(* IEC 61131-3 sources: matiec/tests/cli/profile-fixtures, 26 files *)

(* ---- namespace-internal-local.st ---- *)
NAMESPACE INTERNAL Secret
TYPE
  Value : INT;
END_TYPE

FUNCTION Identity : Value
  VAR_INPUT
    Input : Value;
  END_VAR
  Identity := Input;
END_FUNCTION
END_NAMESPACE

(* ---- reference-local-lifetime.st ---- *)
FUNCTION REFERENCE_LOCAL_LIFETIME_TEST : INT
  VAR
    VALUE : INT;
    VALUE_REF : REF_TO INT;
  END_VAR

  VALUE := 7;
  VALUE_REF := REF(VALUE);
  REFERENCE_LOCAL_LIFETIME_TEST := VALUE_REF^;
END_FUNCTION

(* ---- object-method-nested.st ---- *)
FUNCTION_BLOCK NestedCounter
  VAR Count : INT := 0; END_VAR
  Count := Count;

  METHOD PUBLIC Increment : INT
    VAR_INPUT Delta : INT; END_VAR
    Count := Count + Delta;
    Increment := Count;
  END_METHOD
END_FUNCTION_BLOCK

PROGRAM NestedDemo
  VAR
    Instance : NestedCounter;
    Result : INT;
  END_VAR
  Result := Instance.Increment(Instance.Increment(1));
END_PROGRAM

(* ---- object-method-private.st ---- *)
FUNCTION_BLOCK Counter
  VAR
    Count : INT;
  END_VAR
  Count := Count;

  METHOD PRIVATE Hidden : INT
    Hidden := Count;
  END_METHOD
END_FUNCTION_BLOCK

(* ---- object-method-unknown.st ---- *)
FUNCTION_BLOCK Counter
  VAR
    Count : INT;
  END_VAR
  Count := Count;

  METHOD PUBLIC Increment : INT
    Increment := Count;
  END_METHOD
END_FUNCTION_BLOCK

PROGRAM BadMethod
  VAR
    CounterInstance : Counter;
    Result : INT;
  END_VAR
  Result := CounterInstance.Missing();
END_PROGRAM

(* ---- object-method.st ---- *)
FUNCTION_BLOCK Counter
  VAR
    Count : INT := 0;
  END_VAR

  Count := Count;

  METHOD PUBLIC Increment : INT
    VAR_INPUT
      Delta : INT;
    END_VAR
    VAR
      Amount : INT;
    END_VAR
    Amount := Delta;
    Count := Count + Amount;
    Increment := Count;
  END_METHOD
END_FUNCTION_BLOCK

PROGRAM MethodDemo
  VAR
    CounterInstance : Counter;
    Result : INT;
  END_VAR
  Result := CounterInstance.Increment(Delta := 2);
END_PROGRAM

CONFIGURATION config
  RESOURCE resource1 ON PLC
    TASK main_task(INTERVAL := T#1000ms, PRIORITY := 0);
    PROGRAM instance0 WITH main_task : MethodDemo;
  END_RESOURCE
END_CONFIGURATION

(* ---- semantic-lookup-matrix.st ---- *)
TYPE
  Point : STRUCT X : INT; END_STRUCT;
  PointArray : ARRAY [1..2] OF Point;
END_TYPE

FUNCTION_BLOCK Cell
  VAR Value : INT; END_VAR
  Value := Value;
END_FUNCTION_BLOCK

FUNCTION Adjust : INT
  VAR_INPUT Source : INT; END_VAR
  VAR_OUTPUT Copy : INT; END_VAR
  VAR_IN_OUT Target : INT; END_VAR
  Copy := Source;
  Target := Target + Source;
  Adjust := Target;
END_FUNCTION

PROGRAM LookupMatrix
  VAR
    Item : Point;
    Items : PointArray;
    Block : Cell;
    InputValue : INT;
    OutputValue : INT;
  END_VAR
  Item.X := InputValue;
  Items[1].X := Item.X;
  Block.Value := Items[1].X;
  OutputValue := Adjust(Source := Block.Value, Copy => OutputValue,
                        Target := Items[2].X);
END_PROGRAM

(* ---- assert-invalid.st ---- *)
PROGRAM InvalidAssert
  VAR
    Value : BOOL;
  END_VAR
  Value := ASSERT(Value);
END_PROGRAM

(* ---- assert-multiline.st ---- *)
PROGRAM AssertionFormatting
  VAR
    Ready : BOOL := TRUE;
  END_VAR

  ASSERT (* condition remains ordinary ST *) (
    Ready
  );
END_PROGRAM

(* ---- assert.st ---- *)
PROGRAM AssertDemo
  VAR
    Result : INT;
  END_VAR
  ASSERT(TRUE);
  ASSERT(FALSE);
  Result := 42;
END_PROGRAM

CONFIGURATION config
  RESOURCE resource1 ON PLC
    TASK main_task(INTERVAL := T#1000ms, PRIORITY := 0);
    PROGRAM instance0 WITH main_task : AssertDemo;
  END_RESOURCE
END_CONFIGURATION

(* ---- legacy-assert-function.st ---- *)
FUNCTION ASSERT : BOOL
  VAR_INPUT
    IN : BOOL;
  END_VAR
  ASSERT := IN;
END_FUNCTION

PROGRAM LegacyAssertName
  VAR
    Value : BOOL;
  END_VAR
  Value := ASSERT(TRUE);
END_PROGRAM

(* ---- namespace-ambiguous.st ---- *)
NAMESPACE First
TYPE
  Value : INT;
END_TYPE
END_NAMESPACE

NAMESPACE Second
TYPE
  Value : INT;
END_TYPE
END_NAMESPACE

USING First;
USING Second;

PROGRAM Main
  VAR
    Current : Value;
  END_VAR
END_PROGRAM

(* ---- namespace-internal.st ---- *)
NAMESPACE INTERNAL Secret
TYPE
  Value : INT;
END_TYPE
END_NAMESPACE

PROGRAM Main
  VAR
    Current : Secret.Value;
  END_VAR
END_PROGRAM

(* ---- namespace-using.st ---- *)
NAMESPACE Factory.Motion
TYPE
  Speed : INT;
END_TYPE
END_NAMESPACE

USING Factory.Motion;

PROGRAM Main
  VAR
    Current : Speed := 7;
  END_VAR
  Current := Current;
END_PROGRAM

(* ---- namespace.st ---- *)
NAMESPACE Factory.Motion
TYPE
  Speed : INT;
END_TYPE

FUNCTION Clamp : Speed
  VAR_INPUT
    Value : Speed;
  END_VAR
  Clamp := Value;
END_FUNCTION
END_NAMESPACE

PROGRAM Main
  VAR
    Current : Factory.Motion.Speed := 7;
  END_VAR
  Current := Factory.Motion.Clamp(Current);
END_PROGRAM

(* ---- reference-broad-extension.st ---- *)
TYPE
  REFERENCE_HOLDER : STRUCT
    VALUE_REF : REF_TO INT;
  END_STRUCT;
END_TYPE

PROGRAM REFERENCE_BROAD_EXTENSION_TEST
  VAR
    VALUE : INT;
  END_VAR

  VALUE := VALUE;
END_PROGRAM

(* ---- reference-incompatible.st ---- *)
PROGRAM REFERENCE_INCOMPATIBLE_TEST
  VAR
    REAL_VALUE : REAL;
    INT_REF : REF_TO INT;
  END_VAR

  INT_REF := REF(REAL_VALUE);
END_PROGRAM

(* ---- reference-null.st ---- *)
PROGRAM REFERENCE_NULL_TEST
  VAR
    VALUE : INT;
    VALUE_REF : REF_TO INT := NULL;
  END_VAR

  VALUE_REF := REF(VALUE);
  VALUE := DREF(VALUE_REF);
END_PROGRAM

(* ---- reference.st ---- *)
PROGRAM reference_profile_test
  VAR
    value : INT;
    value_ref : REF_TO INT;
  END_VAR

  value_ref := REF(value);
  value := value_ref^;
END_PROGRAM

(* ---- semantic-duplicate-declaration.st ---- *)
PROGRAM DuplicateDeclaration
  VAR
    Value : INT;
    value : BOOL;
  END_VAR
  Value := 1;
END_PROGRAM

(* ---- semantic-inout-literal.st ---- *)
FUNCTION Bump : INT
  VAR_IN_OUT Target : INT; END_VAR
  Target := Target + 1;
  Bump := Target;
END_FUNCTION

PROGRAM InvalidInOut
  VAR Result : INT; END_VAR
  Result := Bump(1);
END_PROGRAM

(* ---- utf8.st ---- *)
PROGRAM UTF8_SAMPLE
  VAR
    MESSAGE : STRING := '中文🚀';
  END_VAR

  MESSAGE := MESSAGE;
END_PROGRAM

(* ---- var-access-hierarchical-invalid.st ---- *)
TYPE
  IntArray : ARRAY [1..3] OF INT;
  DeviceState : STRUCT
    Value : INT;
  END_STRUCT;
END_TYPE

PROGRAM InvalidAccessProducer
  VAR_OUTPUT
    Value : INT;
  END_VAR
  Value := Value;
END_PROGRAM

CONFIGURATION InvalidHierarchicalAccess
  VAR_GLOBAL
    State : DeviceState;
    Values : IntArray;
  END_VAR
  RESOURCE Resource1 ON PLC
    TASK MainTask(INTERVAL := T#1000ms, PRIORITY := 0);
    PROGRAM Producer WITH MainTask : InvalidAccessProducer;
  END_RESOURCE
  VAR_ACCESS
    MissingField : State.Missing : INT;
    InvalidSelector : State[1] : INT;
    OutsideBounds : Values[4] : INT;
    MissingOutput : Resource1.Producer.Missing : INT;
    WrongType : State.Value : BOOL;
  END_VAR
END_CONFIGURATION

(* ---- var-access-hierarchical.st ---- *)
TYPE
  SampleArray : ARRAY [1..3] OF INT;
  DeviceState : STRUCT
    Value : INT;
    Samples : SampleArray;
  END_STRUCT;
END_TYPE

PROGRAM AccessProducer
  VAR_OUTPUT
    Snapshot : DeviceState;
  END_VAR
  Snapshot.Value := Snapshot.Value;
END_PROGRAM

CONFIGURATION HierarchicalAccessConfig
  VAR_GLOBAL
    State : DeviceState;
    Values : SampleArray;
  END_VAR

  RESOURCE Resource1 ON PLC
    VAR_GLOBAL
      LocalState : DeviceState;
    END_VAR
    TASK MainTask(INTERVAL := T#1000ms, PRIORITY := 0);
    PROGRAM Producer WITH MainTask : AccessProducer;
  END_RESOURCE

  VAR_ACCESS
    ConfigField : State.Value : INT READ_WRITE;
    ConfigArray : Values[2] : INT;
    NestedArray : State.Samples[3] : INT;
    ResourceField : Resource1.LocalState.Value : INT;
    ProgramField : Resource1.Producer.Snapshot.Value : INT;
  END_VAR
END_CONFIGURATION

(* ---- var-access-unresolved.st ---- *)
PROGRAM AccessDemo
  VAR Value : INT; END_VAR
  Value := Value;
END_PROGRAM

CONFIGURATION AccessConfig
  VAR_GLOBAL
    Setpoint : INT;
  END_VAR
  RESOURCE Resource1 ON PLC
    PROGRAM Instance0 : AccessDemo;
  END_RESOURCE
  VAR_ACCESS
    MissingExport : Missing : INT READ_ONLY;
  END_VAR
END_CONFIGURATION

(* ---- var-access.st ---- *)
TYPE
  AccessCount : INT;
END_TYPE

PROGRAM AccessDemo
  VAR
    Value : INT;
  END_VAR
  Value := Value;
END_PROGRAM

CONFIGURATION AccessConfig
  VAR_GLOBAL
    Setpoint : INT := 7;
    Counter : AccessCount := 3;
  END_VAR

  RESOURCE Resource1 ON PLC
    TASK MainTask(INTERVAL := T#1000ms, PRIORITY := 0);
    PROGRAM Instance0 WITH MainTask : AccessDemo;
  END_RESOURCE

  VAR_ACCESS
    RemoteSetpoint : Setpoint : INT READ_WRITE;
    MonitorSetpoint : Setpoint : INT;
    MonitorCounter : Counter : AccessCount;
  END_VAR
END_CONFIGURATION
